PROGRAM AdditionalProgram
VAR
END_VAR

END_PROGRAM

(* stored: Version 1.1.0.1, ProductVersion 3.1.4026.6
   POU AdditionalProgram: Id {c5768f37-9feb-4598-8ecc-00571bc61d8b}, SpecialFunc None *)
